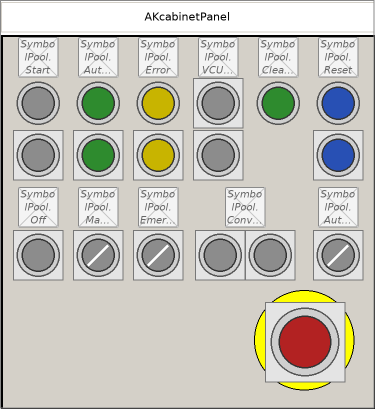
VISUALIZATION V_AKcabinetPanel  // 375x409
VAR_IN_OUT
	Signals : ST_AKcabinetPanel;
END_VAR
    Rectangle (1,35 374x374)
    Lamp1 (13,78 50x50), tooltip "Main contactor activeated", variable: Signals.outputs.LED_MainContactorActivated, style: Lamp-Lamp1-Gray
    PushSwitch (13,130 50x50), tooltip "Activate main contactor", variable: Signals.inputs.PB_ActivateMainContactor, behaviour: TAP, style: Switch-PushSwitch-Gray
    PushSwitch (73,130 50x50), tooltip "Auto on", variable: Signals.inputs.PB_AutoOn, behaviour: TAP, style: Switch-PushSwitch-Green
    Lamp1 (73,78 50x50), tooltip "Auto activated", variable: Signals.outputs.LED_AutoIsOn, style: Lamp-Lamp1-Green
    Lamp1 (133,78 50x50), tooltip "Error", variable: Signals.outputs.LED_Error, style: Lamp-Lamp1-Yellow
    PushSwitch (133,130 50x50), tooltip "Reset error", variable: Signals.inputs.PB_ErrorReset, behaviour: TAP, style: Switch-PushSwitch-Yellow
    RotarySwitch (73,230 50x50), tooltip "Man/Auto key switch", variable: Signals.inputs.SW_Auto, behaviour: TOGGLE, style: Switch-RotarySwitch-Gray
    PushSwitch (13,230 50x50), tooltip "Main contactor off", variable: Signals.inputs.PB_MainContactorOff, behaviour: TAP, style: Switch-PushSwitch-Gray
    Image (18,37 40x40), image: SymbolPool.Start
    Image (78,37 40x40), image: SymbolPool.AutoOn
    Image (138,37 40x40), image: SymbolPool.Error
    Image (18,187 40x40), image: SymbolPool.Off
    Image (78,187 40x40), image: SymbolPool.ManAuto
    Image (198,37 40x40), image: SymbolPool.VCUpDown
    PushSwitch (193,130 50x50), tooltip "VC Down", variable: Signals.inputs.PB_VcDown, behaviour: TAP, style: Switch-PushSwitch-Gray
    PushSwitch (193,78 50x50), tooltip "VC Up", variable: Signals.inputs.PB_VcUp, behaviour: TAP, style: Switch-PushSwitch-Gray
    Lamp1 (253,78 50x50), tooltip "Clear enterance", variable: Signals.outputs.LED_ClearEnterance, style: Lamp-Lamp1-Green
    Lamp1 (313,78 50x50), tooltip "Emergency stop", variable: Signals.outputs.LED_EmergencyStop, style: Lamp-Lamp1-Blue
    PushSwitch (313,130 50x50), tooltip "Reset emergency stop", variable: Signals.inputs.PB_EmergencyStopReset, behaviour: TAP, style: Switch-PushSwitch-Blue
    Image (258,37 40x40), image: SymbolPool.ClearToEnter
    Image (318,37 40x40), image: SymbolPool.Reset
    Image (225,187 40x40), image: SymbolPool.Conv_L_R
    PushSwitch (245,230 50x50), tooltip "VC Conveyor Right", variable: Signals.inputs.PB_VcConvRight, behaviour: TAP, style: Switch-PushSwitch-Gray
    PushSwitch (195,230 50x50), tooltip "VC Conveyor Left", variable: Signals.inputs.PB_VcConvLeft, behaviour: TAP, style: Switch-PushSwitch-Gray
    Image (318,187 40x40), image: SymbolPool.AutoMan
    RotarySwitch (313,230 50x50), tooltip "Auto/Entry request key switch", variable: Signals.inputs.SW_EntryRequest, behaviour: TOGGLE, style: Switch-RotarySwitch-Gray
    RotarySwitch (133,230 50x50), tooltip "Emergency drive key switch", variable: Signals.inputs.SW_EmergencyDrive, behaviour: TOGGLE, style: Switch-RotarySwitch-Gray
    Image (138,187 40x40), image: SymbolPool.EmergencyDrive
    Ellipse (254,290 100x100)
    PushSwitch (265,302 80x80), variable: Signals.inputs.PB_EmergencyStop, behaviour: TOGGLE, style: Switch-PushSwitch-Red
    Textfield (1,2 373x30), "AKcabinetPanel"
END_VISUALIZATION

(* stored: Version 1.1.0.1, ProductVersion 3.1.4024.4
   Visu V_AKcabinetPanel: Id {27c9d086-0fbf-4ef4-a43c-f182601b8f3c} *)
